FUNCTION_BLOCK OUT_MATRIX (* Tabular MATRIX output *)
  (* Standard: 61499-2 *)
  (* Version 0.0, 2004-06-22, JHC, Rockwell Automation *)
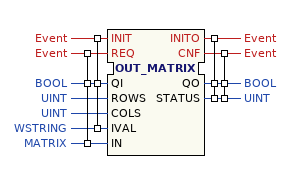
  EVENT_INPUT
    INIT WITH QI, IVAL; (* Initialize matrix from IVAL *)
    REQ WITH QI, IN; (* Write IN to OUT and display *)
  END_EVENT
  EVENT_OUTPUT
    INITO WITH QO, STATUS; (* Initialization Confirm *)
    CNF WITH QO, STATUS; (* Confirmation of REQ *)
  END_EVENT
  VAR_INPUT
    QI : BOOL; (* 1=Enabled,0=Inhibited *)
    ROWS : UINT := 1; (* Initial number of rows in the table *)
    COLS : UINT := 1; (* Initial number of columns in the table *)
    IVAL : WSTRING; (* Initial data values, e.g., "[1,2,3,4]" *)
    IN : MATRIX; (* New value to output *)
  END_VAR
  VAR_OUTPUT
    QO : BOOL; (* 0=OK,1=Inhibited *)
    STATUS : UINT; (* 0=OK,2=TYPE_CONVERSION_ERROR,4=INHIBITED,13=ARRAY_SIZE_ERROR *)
  END_VAR
END_FUNCTION_BLOCK
